// TIA Portal V20 export
DATA_BLOCK "Dummy"   // DB93
{ S7_Optimized_Access := 'TRUE' }
// stored: MemoryReserve 100
   VAR
      RT01 { ExternalAccessible := 'False'; ExternalVisible := 'False'; ExternalWritable := 'False'} : "RT_IF_UDT";
      RT02 { ExternalAccessible := 'False'; ExternalVisible := 'False'; ExternalWritable := 'False'} : "RT_IF_UDT";
      RT03 { ExternalAccessible := 'False'; ExternalVisible := 'False'; ExternalWritable := 'False'} : "RT_IF_UDT";
   END_VAR
BEGIN
END_DATA_BLOCK
